FUNCTION_BLOCK ABSTRACT FB_HE_SATT_Filter IMPLEMENTS I_HE_SATT_Filter
VAR
    iHolder : I_HE_SATT_FilterHolder;
    fLength : LREAL;
    eMaterial : E_HE_SATT_FilterMaterial;
    eStatus : E_HE_SATT_FilterStatus;
END_VAR


METHOD FB_Init: BOOL
VAR_INPUT
    bInitRetains: BOOL; // TRUE: the retain variables are initialized (reset warm / reset cold)
    bInCopyCode: BOOL;  // TRUE: the instance will be copied to the copy code afterward (online change)   
    
    iHolder : I_HE_SATT_FilterHolder;
    fDefaultLength : LREAL;
    eDefaultMaterial : E_HE_SATT_FilterMaterial;
    eDefaultStatus : E_HE_SATT_FilterStatus;
END_VAR

THIS^.iHolder := iHolder;
THIS^.fLength := fDefaultLength;
THIS^.eMaterial := eDefaultMaterial;
THIS^.eStatus := eDefaultStatus;
END_METHOD


PROPERTY Holder : I_HE_SATT_FilterHolder
GET

Holder := THIS^.iHolder;
END_GET
END_PROPERTY


PROPERTY Length : LREAL
GET

Length := THIS^.fLength;
END_GET
SET

THIS^.fLength := Length;
END_SET
END_PROPERTY


PROPERTY Material : E_HE_SATT_FilterMaterial
GET

Material := THIS^.eMaterial;
END_GET
SET

THIS^.eMaterial := Material;
END_SET
END_PROPERTY


PROPERTY MaterialFormula : T_MaxString
GET

MaterialFormula := F_HE_SATT_MaterialToMaterialFormula(eMaterial := THIS^.eMaterial);
END_GET
END_PROPERTY


PROPERTY Status : E_HE_SATT_FilterStatus
GET

Status := THIS^.eStatus;
END_GET
SET

THIS^.eStatus := Status;
END_SET
END_PROPERTY

END_FUNCTION_BLOCK

(* stored: Version 1.1.0.1
   POU FB_HE_SATT_Filter: Id {88a3f423-5332-4112-92bc-be5fb052a1e4}, SpecialFunc None
   Method FB_Init: Id {f9013f92-842c-4d98-883a-911e2061f181}
   Property Holder: Id {84c76333-6b2c-448b-afba-b10d7ed07d24}
   Get Get: Id {d0ad6522-eae7-48b4-99c3-287e93e09af7}
   Property Length: Id {ff7c6bec-3745-4b90-9216-0cfcef73e077}
   Get Get: Id {d297bb58-3c41-4eb0-b6a4-fce9907a9c35}
   Set Set: Id {038089bd-f63d-49ea-acda-2ae7ba207169}
   Property Material: Id {af789a46-91c4-49e3-a56f-f49c20f68172}
   Get Get: Id {b0329835-5996-4837-af01-deefa0300606}
   Set Set: Id {79259363-e825-4934-9c47-7ae0e1080a2d}
   Property MaterialFormula: Id {9821b05d-679a-4604-83c0-ac734674db22}
   Get Get: Id {c51c21c2-fbdc-4482-bed7-37cdb2c1fab5}
   Property Status: Id {57007480-c1de-4d13-9843-5d9e9ffa8744}
   Get Get: Id {7610e0be-6d49-4f72-a1fa-04855866f59c}
   Set Set: Id {3fa0680d-7481-4a03-8cf1-0e6a15b23d1c} *)
